(* CODESYS project SPT_Tracing.library
   Company: Beckhoff Automation LLC
   DefaultNamespace: SPT_Tracing
   Version: 3.0.2
   Placeholder: SPT Tracing
   Title: SPT Tracing

Project tree, tasks and I/O mapping:
  libraries: SPT Base Types, * (Beckhoff Automation LLC); Tc2_EtherCAT, * (Beckhoff Automation GmbH); Tc2_Standard, * (Beckhoff Automation GmbH); Tc2_System, * (Beckhoff Automation GmbH); Tc2_Utilities, * (Beckhoff Automation GmbH); Tc3_EventLogger, * (Beckhoff Automation GmbH); Tc3_JsonXml, * (Beckhoff Automation GmbH)
  Listener/
    function block FB_MessageListener [ST]: Listener, OnMessageSent
    function block FB_TraceListenerBase [ST]: CyclicLogic, Initialize, OnTraceReceived
    interface I_TraceListener: OnTraceReceived
    data type ST_TraceMessage
  Project Information/
    function F_GetCompany [ST]
    function F_GetTitle [ST]
    function F_GetVersion [ST]
  Version/
    global variables Global_Version
  function block FB_TraceLog [ST]: AddContext, AddEntry, AddEntryWithJson, FB_init, TracingAllowed
  global variables Parameters_Tracing
  global variables Tracing
*)

// Listener/ST_TraceMessage
TYPE ST_TraceMessage :
    STRUCT
        Timestamp : T_MaxString;
        Source    : T_MaxString;
        Context   : T_MaxString;
        ScanCount : UDINT;
        Flags     : UDINT;
        Message   : T_MaxString;
        Json      : T_MaxString;
    END_STRUCT
END_TYPE

// Version/Global_Version
{attribute 'TcGenerated'}
{attribute 'no-analysis'}
{attribute 'linkalways'}
// This function has been automatically generated from the project information.
VAR_GLOBAL CONSTANT
	{attribute 'const_non_replaced'}
	stLibVersion_SPT_Tracing : ST_LibVersion := (iMajor := 3, iMinor := 0, iBuild := 2, iRevision := 0, nFlags := 1, sVersion := '3.0.2');
END_VAR

// Parameters_Tracing
{attribute 'qualified_only'}
VAR_GLOBAL CONSTANT
    TRACING_ENABLED          : BOOL  := TRUE;
    MAX_LOG_ENTRIES_PER_SCAN : UDINT := 100;
END_VAR

// Tracing
{attribute 'qualified_only'}
VAR_GLOBAL
    GlobalTraceLog : FB_TraceLog;
END_VAR

// Listener/FB_MessageListener
FUNCTION_BLOCK FINAL FB_MessageListener EXTENDS FB_ListenerBase2
VAR
    Json          : FB_JsonDomParser; //Parse JSON attribute of messages
    JsonAttribute : STRING(10000);    //Holds JSON attribute
    hr            : HRESULT;          //Signals JSON attribute was successfully read
    ipListener    : I_TraceListener;  //Receives callback once message is processed
END_VAR

PROPERTY Listener : I_TraceListener
SET
ipListener := Listener;
END_SET
END_PROPERTY

METHOD OnMessageSent : HRESULT
VAR_INPUT
    fbEvent : REFERENCE TO FB_TcEvent;
END_VAR

VAR
    Message      : ST_TraceMessage;
    JsonDocument : SJsonValue;
    JsonProperty : SJsonValue;
END_VAR
hr := fbEvent.GetJsonAttribute(JsonAttribute, SIZEOF(JsonAttribute));
IF SUCCEEDED(hr) THEN
    JsonDocument := Json.ParseDocument(JsonAttribute);
    IF Json.HasMember(JsonDocument, 'DCTimeStamp') THEN
        JsonProperty      := Json.FindMember(JsonDocument, 'DCTimeStamp');
        Message.Timestamp := Json.GetString(JsonProperty);
    END_IF

    IF Json.HasMember(JsonDocument, 'Instance') THEN
        JsonProperty   := Json.FindMember(JsonDocument, 'Instance');
        Message.Source := Json.GetString(JsonProperty);
    END_IF

    IF Json.HasMember(JsonDocument, 'Context') THEN
        JsonProperty    := Json.FindMember(JsonDocument, 'Context');
        Message.Context := Json.GetString(JsonProperty);
    END_IF

    IF Json.HasMember(JsonDocument, 'ScanCount') THEN
        JsonProperty      := Json.FindMember(JsonDocument, 'ScanCount');
        Message.ScanCount := Json.GetUint(JsonProperty);
    END_IF

    IF Json.HasMember(JsonDocument, 'Flags') THEN
        JsonProperty  := Json.FindMember(JsonDocument, 'Flags');
        Message.Flags := Json.GetUint(JsonProperty);
    END_IF

    IF Json.HasMember(JsonDocument, 'Message') THEN
        JsonProperty    := Json.FindMember(JsonDocument, 'Message');
        Message.Message := Json.GetString(JsonProperty);
    END_IF

    IF Json.HasMember(JsonDocument, 'ExtendedInfo') THEN
        JsonProperty := Json.FindMember(JsonDocument, 'ExtendedInfo');
        Message.Json := Json.GetString(JsonProperty);
    END_IF

    IF ipListener <> 0 THEN
        //Notify listener of message data
        ipListener.OnTraceReceived(Message);
    END_IF
END_IF

OnMessageSent := S_OK; // in order to receive more callbacks (Set <> S_OK in order to cancel the callbacks for this program cycle.)
END_METHOD

END_FUNCTION_BLOCK

// Listener/I_TraceListener
INTERFACE I_TraceListener

METHOD OnTraceReceived
VAR_INPUT
    Message : ST_TraceMessage;
END_VAR
END_METHOD

END_INTERFACE

// Listener/FB_TraceListenerBase
FUNCTION_BLOCK ABSTRACT FB_TraceListenerBase EXTENDS FB_CyclicFB IMPLEMENTS I_TraceListener
VAR_INPUT
END_VAR

VAR_OUTPUT
END_VAR

VAR
    MessageListener : FB_MessageListener;
END_VAR

METHOD PUBLIC CyclicLogic
IF NOT _InitComplete THEN
    _InitComplete := Initialize();
    RETURN;
END_IF

MessageListener.Execute();
END_METHOD

METHOD PROTECTED Initialize : BOOL
VAR
    ListenerFilter : FB_TcEventFilter;
    hr             : HRESULT;
END_VAR
MessageListener.Listener := THIS^;                                   //For callbacks on message received
ListenerFilter.Clear().EventClass.EqualTo(TC_EVENT_CLASSES.Tracing); //Filter events by tracing class
hr := MessageListener.Subscribe2(ListenerFilter);                    //Subscribe to retrieve defined events
IF SUCCEEDED(hr) THEN
    Initialize := TRUE;
END_IF
END_METHOD

METHOD ABSTRACT OnTraceReceived
VAR_INPUT
    Message : ST_TraceMessage;
END_VAR
//Override this method to implement your specific handling
END_METHOD

END_FUNCTION_BLOCK

// Project Information/F_GetCompany
// This function has been automatically generated from the project information.
{attribute 'signature_flag' := '1073741824'}
{attribute 'TcGenerated'}
{attribute 'no-analysis'}
FUNCTION F_GetCompany : WSTRING
VAR_INPUT
	
END_VAR

F_GetCompany := "Beckhoff Automation LLC";

END_FUNCTION

// Project Information/F_GetTitle
// This function has been automatically generated from the project information.
{attribute 'signature_flag' := '1073741824'}
{attribute 'TcGenerated'}
{attribute 'no-analysis'}
FUNCTION F_GetTitle : WSTRING
VAR_INPUT
	
END_VAR

F_GetTitle := "SPT Tracing";

END_FUNCTION

// Project Information/F_GetVersion
// This function has been automatically generated from the project information.
{attribute 'signature_flag' := '1073741824'}
{attribute 'TcGenerated'}
{attribute 'no-analysis'}
FUNCTION F_GetVersion : ST_LibVersion
VAR_INPUT
	
END_VAR

F_GetVersion.iMajor := 3;
F_GetVersion.iMinor := 0;
F_GetVersion.iBuild := 2;
F_GetVersion.iRevision := 0;
F_GetVersion.sVersion := '3.0.2';
F_GetVersion.nFlags := 1;

END_FUNCTION

// FB_TraceLog
FUNCTION_BLOCK FINAL FB_TraceLog
VAR
    Event         : FB_TcMessage;
    JsonParser    : FB_JsonDomParser;
    TimeFormatter : FB_FormatString;
	
	MessagesSentThisScan : UDINT;
END_VAR

METHOD PRIVATE AddContext
VAR_INPUT
    Source  : T_MaxString;
    Flags   : UDINT;
END_VAR

VAR
	CurrentDCTime : DCTIMESTRUCT;
	DCTime100Nsec : WORD;
END_VAR
//Collect DC timestamp info and properly format string
CurrentDCTime := DCTIME64_TO_DCTIMESTRUCT(F_GetActualDcTime64());
DCTime100Nsec := CurrentDCTime.wNanoseconds / 100;
TimeFormatter(sFormat := '%2.2d:%2.2d:%2.2d.%3.3d%3.3d%1.1d',
              arg1    := F_WORD(CurrentDCTime.wHour),
              arg2    := F_WORD(CurrentDCTime.wMinute),
              arg3    := F_WORD(CurrentDCTime.wSecond),
              arg4    := F_WORD(CurrentDCTime.wMilliseconds),
              arg5    := F_WORD(CurrentDCTime.wMicroseconds),
              arg6    := F_WORD(DCTime100Nsec));

Event.ipArguments.AddString(TimeFormatter.sOut);                                                 //DC Timestamp string
Event.ipArguments.AddString(Source);                                                             //POU calling the Trace() function -- this should come automatically
Event.ipArguments.AddString(TwinCAT_SystemInfoVarList._TaskInfo[GETCURTASKINDEXEX()].TaskName);  //Task which called the POU last
Event.ipArguments.AddUDInt(TwinCAT_SystemInfoVarList._TaskInfo[GETCURTASKINDEXEX()].CycleCount); //Cycle count of above task
Event.ipArguments.AddUDInt(Flags);                                                               //General-use flags (application dependent)
END_METHOD

METHOD PUBLIC AddEntry
VAR_INPUT
    Source  : T_MaxString;
    Message : T_MaxString;
    Flags   : UDINT;
END_VAR
{analysis -62}
IF NOT TracingAllowed THEN
	{analysis -90}
    RETURN;
END_IF

Event.ipArguments.Clear().AddString(Message);
AddContext(Source := Source, Flags := Flags);

Event.Send(0);
MessagesSentThisScan := MessagesSentThisScan + 1;
END_METHOD

METHOD PUBLIC AddEntryWithJson
VAR_INPUT
    Source  : T_MaxString;
    Message : T_MaxString;
    Flags   : UDINT;
    Json    : T_MaxString;
END_VAR

VAR
    Document      : SJsonValue;
    JsonAttribute : T_MaxString;
    TaskName      : T_MaxString;
	temp : udint;
END_VAR

VAR_INST
    LastScanCount        : UDINT;
    MessagesSentThisScan : UDINT;
    MissedMessages       : UDINT;
    Throttled            : BOOL;
END_VAR

VAR
    ThrottledNotificationString : T_MaxString;
    CurrentDCTime               : DCTIMESTRUCT;
    DCTime100Nsec               : WORD;
    DCTimeString                : T_MaxString;
END_VAR
{analysis -62}
IF NOT TracingAllowed THEN
    RETURN;
END_IF

Event.ipArguments.Clear().AddString(Message);
AddContext(Source := Source, Flags := Flags);

Document     := JsonParser.NewDocument();
JsonParser.AddJsonMember(Document, 'ExtendedInfo', Json);
JsonAttribute := JsonParser.GetJson(Document);
Event.SetJsonAttribute(JsonAttribute);
Event.Send(0);
MessagesSentThisScan := MessagesSentThisScan + 1;
END_METHOD

METHOD FB_init : BOOL
VAR_INPUT
    bInitRetains : BOOL; // if TRUE, the retain variables are initialized (warm start / cold start)
    bInCopyCode  : BOOL; // if TRUE, the instance afterwards gets moved into the copy code (online change)
END_VAR

VAR
    hr : HRESULT;
END_VAR
{analysis -15}
IF NOT Event.EqualsToEventEntryEx(TC_EVENTS.Tracing.TraceEvent) THEN
    Event.CreateEx(TC_EVENTS.Tracing.TraceEvent, 0);
END_IF
END_METHOD

PROPERTY PRIVATE TracingAllowed : BOOL
GET
VAR_INST
    LastScanCount        : UDINT;
    //MessagesSentThisScan : UDINT;
    MissedMessages       : UDINT;
    Throttled            : BOOL;
END_VAR

VAR
    ThrottledNotificationString : T_MaxString;
END_VAR
{analysis -62}
IF NOT Parameters_Tracing.TRACING_ENABLED THEN
    TracingAllowed := FALSE;
    RETURN;
END_IF

IF TwinCAT_SystemInfoVarList._TaskInfo[GETCURTASKINDEXEX()].CycleCount = LastScanCount THEN
    //Trying to send multiple messages in same scan
    IF Throttled THEN
        MissedMessages := MissedMessages + 1;
        RETURN;
    ELSIF MessagesSentThisScan >= Parameters_Tracing.MAX_LOG_ENTRIES_PER_SCAN AND NOT Throttled THEN
        //Need to throttle messsage queue
        Event.ipArguments.Clear().AddString('Too many messages sent in single scan; tracing throttled.');
        Event.Send(0);
        MissedMessages := MissedMessages + 1;
        Throttled      := TRUE;
        TracingAllowed := FALSE;
        RETURN;
	ELSE
		TracingAllowed := TRUE;
    END_IF
ELSE
    IF Throttled THEN
        ThrottledNotificationString := CONCAT('Missed ', CONCAT(TO_STRING(MissedMessages), ' throttled messages previously.'));
        Event.ipArguments.Clear().AddString(ThrottledNotificationString);
        Event.Send(0);
        MissedMessages := 0;
    END_IF

    LastScanCount        := TwinCAT_SystemInfoVarList._TaskInfo[GETCURTASKINDEXEX()].CycleCount;
    MessagesSentThisScan := 0;
    Throttled            := FALSE;
    TracingAllowed       := TRUE;
END_IF
END_GET
END_PROPERTY

END_FUNCTION_BLOCK
